PROGRAM MAIN
VAR
END_VAR

//resetALL();
XestionModos();						//Chamada a Xestión de Modos
MandoA2Mans(LimiteSoster:=NOT modoAutomatico.goHome);	//Chamada o Mando a 2 mans
gesAlarmas();
IF mandoa2mans.Error THEN
	modoautomatico.goHome:=TRUE;
END_IF
//Se estamos en modo automático chamamos o programa
IF VariablesGlobales.ModoMaquina=modos.Auto THEN
	ModoAutomatico(bOrdenMarcha:=MandoA2Mans.Q,
	bSimular:=VariablesGlobales.Simular,
	ordenhome := io.pulsador1);	
END_IF

END_PROGRAM

(* stored: Version 1.1.0.1, ProductVersion 3.1.4024.9
   POU MAIN: Id {73412b68-e04a-4daa-85d8-3dacf260287a}, SpecialFunc None *)
